TYPE "Positioning_MOL_Machine_Manager"
VERSION : 0.1
// Block: Positioning_MOL_Machine_Manager
   STRUCT
      EnableStopDoorOpeningReq : Bool;
      EnableStopInPhase : Bool;
      EnableStopProgrammed : Bool;
      Control_ON : Bool;
      Minus : Bool;
      Plus : Bool;
      MoveToPos : Bool;
      Pos : LReal;
   END_STRUCT;

END_TYPE
